Fanuc KAREL source: KS00016.KL

PROGRAM KS00016
%NOLOCKGROUP
TYPE
  REC_T = STRUCTURE
    VALUE: INTEGER
    FLAG: BOOLEAN
  ENDSTRUCTURE
VAR
  A: FILE
  B: FILE
  FLAG: BOOLEAN
  N: INTEGER
  STATUS: INTEGER
  PN: STRING[80]
  VN: STRING[80]
BEGIN
  PN = ''
  VN = 'A'
  FLAG = A <> B
END KS00016
